# EPICS substitutions: modules/event/evrSupport/Db/ioc/IOC-LI21-BP01evr.substitutions
#==============================================================================
#
# Abs:  LCLS EVR IOC records for LI21 BP01
#
# Name: IOC-LI21-BP01evr.substitutions
#
#==============================================================================
#
file evrBPXX.db
{
pattern { DEVICE        }
	{ EVR:LI21:BP01 }
}
